# EPICS autosave request: iocProsilica/setupMenu.req
file "configMenu.req",            P=$(P),  CONFIG=$(CONFIG)
file "auto_settings.req", P=$(P)
